FUNCTION_BLOCK C_BINARYWRITER
VAR_INPUT
END_VAR
VAR_OUTPUT
END_VAR
VAR
	_BASESTREAM 	: I_STREAM;
END_VAR

PROPERTY BaseStream : I_STREAM
GET
BaseStream := _BASESTREAM;
END_GET
END_PROPERTY

METHOD Close : DINT
VAR_INPUT
END_VAR
Close := _BASESTREAM.Close();
_BASESTREAM := 0;
RETURN;
END_METHOD

METHOD New : DINT
VAR_INPUT
	STREAM : I_STREAM;
END_VAR
IF STREAM = 0 THEN
	New := 1;
	RETURN;
ELSE
	IF STREAM.IsValid THEN
		_BASESTREAM := STREAM;
		_BASESTREAM.Seek( 0, E_STREAMSEEKTYPE.Origin);
		New := -1;
		RETURN;
	ELSE
		New := 1;
		RETURN;
	END_IF
END_IF
END_METHOD

METHOD Reset : DINT
VAR_INPUT
END_VAR
_BASESTREAM 	:= 0;
Reset := -1;
END_METHOD

METHOD WriteBool : DINT
VAR_INPUT
	in_data : BOOL;
END_VAR
IF _BASESTREAM = 0 THEN
	WriteBool := 1;
	RETURN;
END_IF

WriteBool := _BASESTREAM.Write(ADR(in_data), 1);
RETURN;
END_METHOD

METHOD WriteBytes : DINT
VAR_INPUT
	in_data 	: POINTER TO BYTE;
	length		: UDINT;
END_VAR
IF _BASESTREAM = 0 THEN
	WriteBytes := 1;
	RETURN;
END_IF

WriteBytes := _BASESTREAM.Write(in_data, length);
RETURN;
END_METHOD

METHOD WriteDouble : DINT
VAR_INPUT
	in_data : LREAL;
END_VAR
IF _BASESTREAM = 0 THEN
	WriteDouble := 1;
	RETURN;
END_IF

WriteDouble := _BASESTREAM.Write(ADR(in_data), 8);
RETURN;
END_METHOD

METHOD WriteFloat : DINT
VAR_INPUT
	in_data : REAL;
END_VAR
IF _BASESTREAM = 0 THEN
	WriteFloat := 1;
	RETURN;
END_IF

WriteFloat := _BASESTREAM.Write(ADR(in_data) , 4);
RETURN;
END_METHOD

METHOD WriteInt16 : DINT
VAR_INPUT
	in_data : INT;
END_VAR
IF _BASESTREAM = 0 THEN
	WriteInt16 := 1;
	RETURN;
END_IF

WriteInt16 := _BASESTREAM.Write(ADR(in_data) , 2);
RETURN;
END_METHOD

METHOD WriteInt32 : DINT
VAR_INPUT
	in_data : DINT;
END_VAR
IF _BASESTREAM = 0 THEN
	WriteInt32 := 1;
	RETURN;
END_IF

WriteInt32 := _BASESTREAM.Write(ADR(in_data) , 4);
RETURN;
END_METHOD

METHOD WriteString : DINT
VAR_INPUT
	in_data 	: PVOID;
	length		: UDINT;
END_VAR
IF _BASESTREAM = 0 THEN
	WriteString := 1;
	RETURN;
END_IF

WriteString := _BASESTREAM.Write(in_data, length);
RETURN;
END_METHOD

METHOD WriteUInt16 : DINT
VAR_INPUT
	in_data : UINT;
END_VAR
IF _BASESTREAM = 0 THEN
	WriteUInt16 := 1;
	RETURN;
END_IF

WriteUInt16 := _BASESTREAM.Write(ADR(in_data) , 4);
RETURN;
END_METHOD

METHOD WriteUInt32 : DINT
VAR_INPUT
	in_data : UDINT;
END_VAR
IF _BASESTREAM = 0 THEN
	WriteUInt32 := 1;
	RETURN;
END_IF

WriteUInt32 := _BASESTREAM.Write(ADR(in_data) , 4);
RETURN;
END_METHOD

END_FUNCTION_BLOCK

(* stored: Version 1.1.0.1, ProductVersion 3.1.4019.2
   POU C_BINARYWRITER: Id {e7f30169-cf04-41d2-b79c-23b5695cf795}, SpecialFunc None
   Property BaseStream: Id {3dcd12a4-e306-49ed-938a-5220871db64f}
   Get Get: Id {85b4857b-a5ab-4898-8488-7d4e7f67ebe9}
   Method Close: Id {af4be7ee-df55-43f8-882b-81de066d5a72}
   Method New: Id {bf9e58ea-41d9-42ca-a471-045ce927c089}
   Method Reset: Id {9859fed2-aa19-4a86-9ca2-60f339f48c16}
   Method WriteBool: Id {7743df79-e2d5-49de-99a2-359a2ae83fbb}
   Method WriteBytes: Id {c5f6e455-1e48-420b-aadf-1ba979cd59eb}
   Method WriteDouble: Id {fc137834-c546-4ead-91d9-c3027d0be7cc}
   Method WriteFloat: Id {8d1e632b-d11a-42b0-8774-953d07c3b7e8}
   Method WriteInt16: Id {15bcfc73-e915-4034-a81f-7f040d017fa0}
   Method WriteInt32: Id {904892c4-4133-4397-a7df-060fbc4a953e}
   Method WriteString: Id {7115c34f-7f55-4080-97ae-652a8e87cc88}
   Method WriteUInt16: Id {55423954-4581-4831-bdfd-662fd3d0727d}
   Method WriteUInt32: Id {6ec8e28c-8c95-4b09-a9e3-dca4cf6121f6} *)
